(* IEC 61131-3 sources: Industry-PLC-LLM/data/PLCBEAD_repo/PLCBEAD_PLCEmbed-main/PLC-BEAD/Source/GEB/TIME_TO_DWORD, 1 file *)

(* ---- TIME_TO_DWORD.ST ---- *)
FUNCTION TIME_TO_DWORD1:DWORD

VAR_INPUT
	X :	TIME;
END_VAR

TIME_TO_DWORD1 := UDINT_TO_DWORD(DINT_TO_UDINT(TIME_TO_DINT(X)));
END_FUNCTION

PROGRAM program0
  VAR
	X :	TIME;
    CEIL5_OUT : DWORD;
  END_VAR

  CEIL5_OUT := TIME_TO_DWORD1(X);
END_PROGRAM
